KUKA KRL program: GEARS.src, GEARS.dat

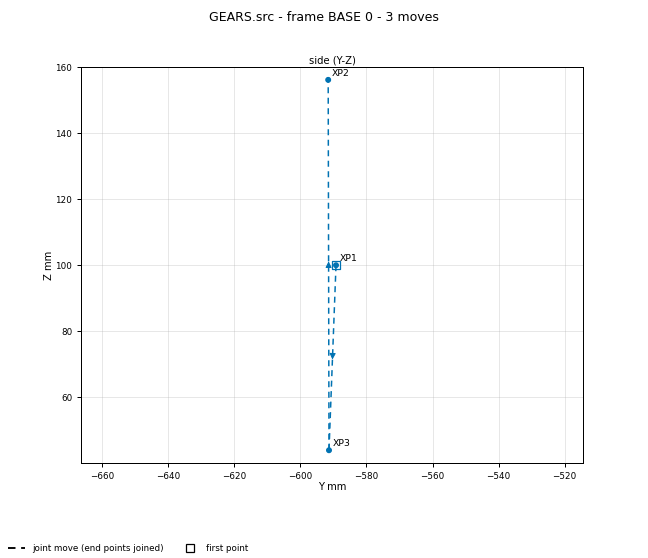
[picture p0: tool path of GEARS.src in frame BASE 0, 3 of 3 moves have a stored position in this frame; points joined in program order, loops and branches not executed]
--- GEARS.src ---
&ACCESS RVP
&REL 62
&PARAM TEMPLATE = C:\KRC\Roboter\Template\vorgabe
&PARAM EDITMASK = *
DEF GEARS( )
DECL FRAME PT1
DECL BOOL TEMP
DECL BOOL STATE
DECL IPO_MODE LAST_IPO
DECL E6POS POSITION
;FOLD INI
  ;FOLD BASISTECH INI
    GLOBAL INTERRUPT DECL 3 WHEN $STOPMESS==TRUE DO IR_STOPM ( )
    INTERRUPT ON 3
    BAS (#INITMOV,0 )
  ;ENDFOLD (BASISTECH INI)
  ;FOLD USER INI
    ;Make your modifications here

  ;ENDFOLD (USER INI)
;ENDFOLD (INI)

$TOOL=TOOL_DATA[5]
$VEL.CP=.2
$VEL.ORI1=100
$VEL.ORI2=100
$ACC.CP=1.0
$ACC.ORI1=80
$ACC.ORI2=80
$ADVANCE=5

;FOLD PTP P1 Vel=100 % PDAT1 Tool[5]:Pneumatic_gripper_probe Base[0];%{PE}%R 5.6.11,%MKUKATPBASIS,%CMOVE,%VPTP,%P 1:PTP, 2:P1, 3:, 5:100, 7:PDAT1
$BWDSTART=FALSE
PDAT_ACT=PPDAT1
FDAT_ACT=FP1
BAS(#PTP_PARAMS,100)
PTP XP1
;ENDFOLD

;PTP{X 11.82,Y -590.80,Z 100,A 3.52,B 0,C -180}

;FOLD PTP P3 Vel=100 % PDAT3 Tool[5]:Pneumatic_gripper_probe Base[0];%{PE}%R 5.6.11,%MKUKATPBASIS,%CMOVE,%VPTP,%P 1:PTP, 2:P3, 3:, 5:100, 7:PDAT3
$BWDSTART=FALSE
PDAT_ACT=PPDAT3
FDAT_ACT=FP3
BAS(#PTP_PARAMS,100)
PTP XP3
;ENDFOLD

STATE = STARTIMPEDANCE(TRUE)
TEMP=SETFORCE("Z",5)

LIN_REL{Z -12}

;LAST_IPO = $IPO_MODE
;$IPO_MODE = #TCP

; Clear all search parameters
STATE = CANCEL_SEARCH()

; Alarm clock test:  Passed
STATE = STATE AND ADDTERMCLOCK(#ALARMCLOCK, #FAIL, 20000.0, 5)

STATE = STATE AND ADDTERMDISTANCE(#SUCCESS, 0.0, 0.0, 20.0,20.0)

;BOOL ADDSEARCHROTATION(REAL RANGE, REAL SPEED)
STATE = STATE AND ADDSEARCHROTATION(60.0, 10.0)

;POSITION=$POS_ACT_MES
WHILE STATE
   STATE = (SEARCH()==#RUNNING)

ENDWHILE

TEMP=FORCEZSTOP()
$STIFFNESS.STRATEGY=10
$STIFFNESS.COMMIT=TRUE

STATE=STARTIMPEDANCE(FALSE)

STATE = CANCEL_SEARCH()

LIN_REL{Z 50}
;FOLD PTP P2 Vel=100 % PDAT2 Tool[5]:Pneumatic_gripper_probe Base[0];%{PE}%R 5.6.11,%MKUKATPBASIS,%CMOVE,%VPTP,%P 1:PTP, 2:P2, 3:, 5:100, 7:PDAT2
$BWDSTART=FALSE
PDAT_ACT=PPDAT2
FDAT_ACT=FP2
BAS(#PTP_PARAMS,100)
PTP XP2
;ENDFOLD


END

--- GEARS.dat ---
&ACCESS RVP
&REL 62
&PARAM TEMPLATE = C:\KRC\Roboter\Template\vorgabe
&PARAM EDITMASK = *
DEFDAT  GEARS
;FOLD EXTERNAL DECLARATIONS;%{PE}%MKUKATPBASIS,%CEXT,%VCOMMON,%P
;FOLD BASISTECH EXT;%{PE}%MKUKATPBASIS,%CEXT,%VEXT,%P
EXT  BAS (BAS_COMMAND  :IN,REAL  :IN )
DECL INT SUCCESS
;ENDFOLD (BASISTECH EXT)
;FOLD USER EXT;%{E}%MKUKATPUSER,%CEXT,%VEXT,%P
;Make here your modifications

;ENDFOLD (USER EXT)
;ENDFOLD (EXTERNAL DECLARATIONS)
DECL BASIS_SUGG_T LAST_BASIS={POINT1[] "P3                      ",POINT2[] "P3                      ",CP_PARAMS[] "CPDAT0                  ",PTP_PARAMS[] "PDAT3                   ",CONT[] "                        ",CP_VEL[] "2.0                     ",PTP_VEL[] "100                     ",SYNC_PARAMS[] "SYNCDAT                 ",SPL_NAME[] "S0                      "}
DECL PDAT PPDAT0={VEL 100.0,ACC 100.0,APO_DIST 100.0,APO_MODE #CPTP}
DECL E6POS XP0={X 12.30126,Y -591.60022,Z 156.144394,A 1.17926598,B -0.00117073196,C -179.9776,S 1,T 36,E1 -0.0129604302,E2 0.0,E3 0.0,E4 0.0,E5 0.0,E6 0.0}
DECL FDAT FP0={TOOL_NO 5,BASE_NO 0,IPO_FRAME #BASE,POINT2[] " ",TQ_STATE FALSE}
DECL PDAT PPDAT1={VEL 100.0,ACC 100.0,APO_DIST 100.0,APO_MODE #CPTP}
DECL E6POS XP1={X 11.8614197,Y -589.22699,Z 99.9752121,A 0.00196523895,B -0.000274408609,C -179.9935,S 1,T 44,E1 0.354849786,E2 0.0,E3 0.0,E4 0.0,E5 0.0,E6 0.0}
DECL FDAT FP1={TOOL_NO 5,BASE_NO 0,IPO_FRAME #BASE,POINT2[] " ",TQ_STATE FALSE}
DECL PDAT PPDAT2={VEL 100.0,ACC 100.0,APO_DIST 100.0,APO_MODE #CPTP}
DECL E6POS XP2={X 12.3132296,Y -591.593079,Z 156.112793,A 1.184057,B -0.00175605796,C -179.975296,S 1,T 36,E1 -0.0125227002,E2 0.0,E3 0.0,E4 0.0,E5 0.0,E6 0.0}
DECL FDAT FP2={TOOL_NO 5,BASE_NO 0,IPO_FRAME #BASE,POINT2[] " ",TQ_STATE FALSE}
DECL E6POS XP3={X 11.9817305,Y -591.349182,Z 43.9423599,A -2.7256999,B -0.438843489,C 179.203003,S 1,T 44,E1 1.45612597,E2 0.0,E3 0.0,E4 0.0,E5 0.0,E6 0.0}
DECL FDAT FP3={TOOL_NO 5,BASE_NO 0,IPO_FRAME #BASE,POINT2[] " ",TQ_STATE FALSE}
DECL PDAT PPDAT3={VEL 100.0,ACC 100.0,APO_DIST 100.0,APO_MODE #CPTP}
ENDDAT
